// TIA Portal V16 export
// export: Created 2021-06-20T01:36:49.7692502Z, ExportSetting WithDefaults, DisplayName Totally Integrated Automation Portal, DisplayVersion V16 Update 4, DisplayName TIA Portal Version Control Interface, DisplayVersion V16 Update 2, DisplayName TIA Portal Openness, DisplayVersion V16 Update 4, DisplayName STEP 7 Professional, DisplayVersion V16 Update 4, DisplayName STEP 7 Safety, DisplayVersion V16, DisplayName WinCC Advanced, DisplayVersion V16 Update 4
FUNCTION "UserSet" : Void   // FC3, F_FBD
{ S7_Optimized_Access := 'TRUE' }
VERSION : 0.1
// stored: AutoNumber true, IsIECCheckEnabled false, UDAEnableTagReadback false
   VAR_INPUT
      q : Bool;
   END_VAR
   VAR_IN_OUT
      "a" : Bool;
   END_VAR
BEGIN

REGION Network 1
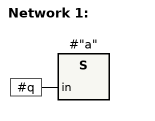
   IF #q THEN #"a" := TRUE; END_IF;
END_REGION
END_FUNCTION
